TYPE ATV212Control :
STRUCT
	bStart		: BOOL;
	bStop		: BOOL;
	bForward	: BOOL;
	fFrequency	: REAL;
END_STRUCT
END_TYPE

(* stored: Version 1.1.0.1, ProductVersion 3.1.4022.18
   DUT ATV212Control: Id {7a1a5339-fdb0-4a22-91a1-40077d67044c} *)
